FUNCTION FC_PMCAlarmToBoolArray : BOOL
VAR_INPUT
	RegA : POINTER TO BYTE;
END_VAR
VAR_OUTPUT
	AlarmList : ARRAY[0..CNC.NUM_MAX_STATION_ALARMS-1] OF BOOL;
END_VAR
VAR
	i : LWORD;
	j : DINT;
	reg: BYTE;
END_VAR

FOR i:= 0 TO 9 DO
	FOR j := 0 TO 7 DO
        AlarmList[(i*8) + j] := TO_BOOL(PBYTE_TO_BYTE((RegA+i)) AND SHL(1,j));
    END_FOR
END_FOR

END_FUNCTION

(* stored: Version 1.1.0.1, ProductVersion 3.1.4024.13
   POU FC_PMCAlarmToBoolArray: Id {f0cefe91-5756-458e-9a50-968dc4d014a6}, SpecialFunc None *)
